{attribute 'GeneratedUsingTerminal: EK1100-0000-0018'}
{attribute addProperty BoxType "EK1100-0000-0018"}
{attribute addProperty Id "Beckhoff_ELM35xxEK1122Beckhoff_ELM35xxEK1122_E14BC85D2A_0001_ELM3502_0000_0016ELM3502_73CCAB7A50A_0002_ELM3502_0000_0017ELM3502_73CCAB7A50A_0003_ELM3502_0000_0018ELM3502_73CCAB7A50A_0004_ELM3502_0000_0019ELM3502_73CCAB7A50A_0005_ELM3504_0000_0016ELM3504_7474644C72A_0006_ELM3504_0000_0017ELM3504_7474644C72A_0007_ELM3504_0000_0018ELM3504_7474644C72A_0008_ELM3504_0000_0019ELM3504_7474644C72"}
{attribute addProperty CRC "568526005"}
{attribute addProperty Size "490"}
TYPE Beckhoff_ELM35xx_21E304B5 EXTENDS EK1100_AB5A9467 :
STRUCT
	{attribute addProperty Name "Beckhoff_ELM35xxEK1122"}
	Beckhoff_ELM35xxEK1122 : Beckhoff_ELM35xxEK1122_E14BC85D;
	{attribute addProperty Name "A_0001_ELM3502_0000_0016"}
	A_0001_ELM3502_0000_0016 : ELM3502_73CCAB7A;
	{attribute addProperty Name "A_0002_ELM3502_0000_0017"}
	A_0002_ELM3502_0000_0017 : ELM3502_73CCAB7A;
	{attribute addProperty Name "A_0003_ELM3502_0000_0018"}
	A_0003_ELM3502_0000_0018 : ELM3502_73CCAB7A;
	{attribute addProperty Name "A_0004_ELM3502_0000_0019"}
	A_0004_ELM3502_0000_0019 : ELM3502_73CCAB7A;
	{attribute addProperty Name "A_0005_ELM3504_0000_0016"}
	A_0005_ELM3504_0000_0016 : ELM3504_7474644C;
	{attribute addProperty Name "A_0006_ELM3504_0000_0017"}
	A_0006_ELM3504_0000_0017 : ELM3504_7474644C;
	{attribute addProperty Name "A_0007_ELM3504_0000_0018"}
	A_0007_ELM3504_0000_0018 : ELM3504_7474644C;
	{attribute addProperty Name "A_0008_ELM3504_0000_0019"}
	A_0008_ELM3504_0000_0019 : ELM3504_7474644C;
END_STRUCT
END_TYPE

(* stored: Version 1.2.0.0, ProductVersion 3.1.4024.9
   DUT Beckhoff_ELM35xx_21E304B5: Id {1782e0fa-7c4f-4edc-8035-bd305458f8e3} *)
